(*~
<docu>
<summary>
	Provides a mechanism for inspecting status of discrete signal.	
</summary>
</docu>
~*)
FUNCTION_BLOCK TcoDataInspector EXTENDS TcoInspector
VAR
    _data : TcoDataInspectorData;
	{attribute 'hide'}
	_lastOutValue : STRING;
END_VAR

(*~
<docu>
<summary>
	Gets data of this inspector.
</summary>
</docu>
~*)
PROPERTY Data : REFERENCE TO TcoDataInspectorData
GET
Data REF= _data;
END_GET
END_PROPERTY

(*~
<docu>
<summary>
	Inspects the signal and evaluates that it matches the value set in `RequiredStatus`.
</summary>
<returns>
	Returns the interface with information about the state of inspection.
</returns>
</docu>
~*)
METHOD Inspect : IInspector
VAR_INPUT
    Status : STRING(255);
END_VAR

VAR
	tmpResult : BOOL;
	charIndex : INT;
	charRequired : STRING(1);
	charAcquired : STRING(1);	
END_VAR

VAR CONSTANT
    epsilon : REAL := 1;
END_VAR
Inspect := THIS^;

OnEnterInspection();

_inspectionData REF= _data;

Invoke();

IF (Execute()) THEN
    IF (_data.IsByPassed) THEN
        _data.Result    := eInspectorResult.Bypassed;
        _data.TimeStamp := Context.RealTimeClock.NowLocal();
        DoneWhen(TRUE);
        RETURN;
    END_IF

		THIS^.Messenger.OnCondition(LEN(Status) > 250 OR LEN(_data.RequiredStatus) > 250).Build().Append('The checked input string or required pattern string exceeds 250 characters.').As().AsError();
		
        IF(LEN(Status) > 250 OR LEN(_data.RequiredStatus) > 254) THEN                
            RETURN;
        END_IF
		
	    _data.DetectedStatus := Status;
		
		
		IF(_data.StarNotationEnabled) THEN
			tmpResult := TRUE;
			FOR charIndex := 1 TO LEN(_data.RequiredStatus) DO
				charRequired := MID(_data.RequiredStatus, 1, charIndex);
				
				IF(LEN(_data.DetectedStatus) >= charIndex) THEN
					charAcquired :=  MID(_data.DetectedStatus, 1, charIndex);
				ELSE
					charAcquired := '';
				END_IF;	
				
				IF(charRequired <> '*' AND charRequired <> '#') THEN
					tmpResult := charRequired = charAcquired;
				ELSIF(charRequired = '#') THEN
					tmpResult := IsNumber(charAcquired);            	
				END_IF
				
				IF(NOT tmpResult) THEN
					EXIT;
				END_IF				
			END_FOR
		ELSE
			
			tmpResult := F_RTrim(_data.DetectedStatus) =F_RTrim(_data.RequiredStatus);	
		END_IF
		
       
		IF(NOT tmpResult) THEN	
			_lastOutValue := Status;
		END_IF
		
		_failTimer(IN:= TRUE, PT:=_data.FailTime);
		_passTimer(IN:= tmpResult,PT:=_data.PassTime);
									  
     	DoneWhen(_failTimer.Q OR _passTimer.Q);
END_IF;
END_METHOD

METHOD PROTECTED IsNumber : BOOL
VAR_INPUT
    inCharacter : STRING(1);
END_VAR
VAR
    numericalRapresentation : BYTE;
END_VAR
IF (inCharacter = '0'
OR  inCharacter = '1'
OR  inCharacter = '2'
OR  inCharacter = '3'
OR  inCharacter = '4'
OR  inCharacter = '5'
OR  inCharacter = '6'
OR  inCharacter = '7'
OR  inCharacter = '8'
OR  inCharacter = '9') 
THEN
	IsNumber := TRUE;
	RETURN;
END_IF;

IsNumber := FALSE;
END_METHOD

(*~
	<docu>
		<summary>
			Executes when task reaches the ```Done``` state .
		</summary>			
	</docu>	
~*)
METHOD PROTECTED OnDone
SUPER^.OnDone();
IF (_data.Result = eInspectorResult.Failed) THEN
     _data.DetectedStatus := _lastOutValue;
END_IF
END_METHOD

END_FUNCTION_BLOCK

(* stored: Version 1.1.0.1, ProductVersion 3.1.4024.9
   POU TcoDataInspector: Id {a28e1549-36e0-0a83-2425-0582897b0a9d}, SpecialFunc None
   Property Data: Id {b0476b77-184e-090e-084e-b715aa910f21}
   Get Get: Id {735a50fd-db59-0580-13ce-a7dea298b20e}
   Method Inspect: Id {f50ce6ff-4be8-058f-29dc-b37b975fecf2}
   Method IsNumber: Id {06fdee84-4be9-0485-30d1-946d69a2763b}
   Method OnDone: Id {2e401878-44db-0db3-3b4e-da671280d16c} *)
